(* IEC 61131-3 sources: com.logicals.lc3.webinar/usRTS_RPMControl_iSOC/src_FB_LIB_SAFE/Safe/Select, 2 files *)

(* ---- wSEL_SAFEBOOL.iecst ---- *)
NAMESPACE logicals.web.standard.safe
NAMESPACE select

/*
 * Function block wrapper for IEC 61131-3 SEL<br>
 * G = selector (SAFEBOOL)<br>
 * IN0 = first value (SAFEBOOL)<br>
 * IN1 = second value (SAFEBOOL)<br>
 * OUT := G ? IN1 : IN0; (SAFEBOOL)<br>
 */
FUNCTION_BLOCK wSEL_SAFEBOOL
	{ vNameAlignment:="center"; altName:="SEL"; bgColor:="Gold"; width:=120; }
	VAR_INPUT
		G : SAFEBOOL;
		IN0 : SAFEBOOL;
		IN1 : SAFEBOOL;
	END_VAR
	VAR_OUTPUT
		OUT : SAFEBOOL;
	END_VAR

	IF (SEL_BOOL(G:=G<>SAFEBOOL_Constant#SAFEFALSE, IN0:=IN0<>SAFEBOOL_Constant#SAFEFALSE, IN1:=IN1<>SAFEBOOL_Constant#SAFEFALSE, ENO=>ENO) <> FALSE)
	THEN
		OUT := SAFEBOOL_Constant#SAFETRUE;
	ELSE
		OUT := SAFEBOOL_Constant#SAFEFALSE;
	END_IF;
	ENO := ENO AND CheckSAFEBOOL(G) AND CheckSAFEBOOL(IN0) AND CheckSAFEBOOL(IN1);
END_FUNCTION_BLOCK

END_NAMESPACE
END_NAMESPACE

(* ---- wSEL_SAFEINT.iecst ---- *)
NAMESPACE logicals.web.standard.safe
NAMESPACE select

/*
 * Function block wrapper for IEC 61131-3 SEL<br>
 * G = selector (SAFEBOOL)<br>
 * IN0 = first value (SAFEINT)<br>
 * IN1 = second value (SAFEINT)<br>
 * OUT := G ? IN1 : IN0; (SAFEINT)<br>
 */
FUNCTION_BLOCK wSEL_SAFEINT
	{ vNameAlignment:="center"; altName:="SEL"; bgColor:="GoldenRod"; width:=120; }
	VAR_INPUT
		G : SAFEBOOL;
		IN0 : SAFEINT;
		IN1 : SAFEINT;
	END_VAR
	VAR_OUTPUT
		OUT : SAFEINT;
	END_VAR

	OUT := SEL_INT(G:=G<>SAFEBOOL_Constant#SAFEFALSE, IN0:=IN0, IN1:=IN1, ENO=>ENO);
	ENO := ENO AND CheckSAFEBOOL(G);
END_FUNCTION_BLOCK

END_NAMESPACE
END_NAMESPACE
